// Mitsubishi GX Works2 project: 22APRIL   PLC: FX3G
// PLC project

// global labels: Global1
VAR_GLOBAL
  Work_Day_Light AT X007 : BOOL;
  Chocolate_First_Input AT D1550 : REAL;
  Chocolate_Stock AT D1350 : REAL;
  Nuts_First_Input AT D1600 : REAL;
  Nuts_Stock AT D1400 : REAL;
  Start_Day AT X007 : BOOL;
  Start AT Y007 : BOOL;
  WorkingDay AT Y007 : BOOL;
  Emergancy AT X005 : BOOL;
  Working_Day_Light AT Y007 : BOOL;
  End_Day AT M1 : BOOL;
  No_Inventory AT M2 : BOOL;
  Pistachio_First_Input AT D1700 : REAL;
  Kadaif_First_Input AT D1650 : REAL;
  Pistachio_Stock AT D1450 : REAL;
  Kadaif_Stock AT D1500 : REAL;
  Melting_Button AT X001 : BOOL;
END_VAR
VAR_GLOBAL CONSTANT
  Chocolate_Amout_Melting : REAL := 400;
END_VAR
VAR_GLOBAL
  No_Choclate AT M3 : BOOL;
  Melting_Light AT Y001 : BOOL;
  Temp_Sensor AT X002 : BOOL;
  Valid_Chocolate AT M11 : BOOL;
  No_Valid_Chocolate AT M11 : BOOL;
  Choose_Filling AT X004 : BOOL;
  Choose_Type_Analog_Input AT D8280 : INT;
END_VAR
VAR_GLOBAL CONSTANT
  const400 : REAL := 400.0;
END_VAR
VAR_GLOBAL
  Real_Undivided_Input AT D1150 : REAL;
  Real_Input AT D1250 : REAL;
  Choose_Type AT X004 : BOOL;
END_VAR
VAR_GLOBAL CONSTANT
  Constant_6 : REAL := 6;
END_VAR
VAR_GLOBAL
  Dubai_Light AT M8 : BOOL;
END_VAR
VAR_GLOBAL CONSTANT
  Constant_5 : REAL := 5;
END_VAR
VAR_GLOBAL
  Nuts_Light AT M9 : BOOL;
  Finished_Packages AT M10 : BOOL;
  Finished_Chocolate_Bar AT CC1 : BOOL;
END_VAR
VAR_GLOBAL CONSTANT
  NutsDubaiAmount : REAL := 20;
  PistachioDubaiAmount : REAL := 120;
  KadaifDubaiAmount : REAL := 60;
END_VAR
VAR_GLOBAL
  Kadai_Stock AT D1500 : REAL;
  Valid_Dubai AT M11 : BOOL;
END_VAR
VAR_GLOBAL CONSTANT
  NutsNutsAmount : REAL := 100;
  PistachioNutsAmount : REAL := 100;
END_VAR
VAR_GLOBAL
  Valid_Nuts AT M12 : BOOL;
END_VAR
VAR_GLOBAL CONSTANT
  ChocolatePackageAmount : REAL := 400;
  Chocolate_Amount_Melting : REAL := 400;
END_VAR
VAR_GLOBAL
  Melting_Container AT D1200 : REAL;
  Loction_Sensor AT X003 : BOOL;
  Constant_4 AT D8280 : INT;
END_VAR
VAR_GLOBAL CONSTANT
  const4 : INT := 40;
END_VAR
VAR_GLOBAL
  Casting_Answer AT TS2 : BOOL;
  Casting AT Y002 : BOOL;
END_VAR
VAR_GLOBAL CONSTANT
  timer4 : REAL := 4;
  const40 : INT := 40;
END_VAR
VAR_GLOBAL
  Filling_Container AT D1800 : REAL;
END_VAR
VAR_GLOBAL CONSTANT
  Dubai_Filling_Total : REAL := 200;
END_VAR
VAR_GLOBAL
  Filling AT M14 : BOOL;
  Flicker AT M6 : BOOL;
  Flicker3 AT TC4 : BOOL;
END_VAR
VAR_GLOBAL CONSTANT
  const50 : INT := 50;
END_VAR
VAR_GLOBAL
  Flicker_Timer3 AT TS4 : BOOL;
  FlickerLight3 AT Y003 : BOOL;
  Flicker4 AT TC5 : BOOL;
  Flicker_Timer4 AT TS5 : BOOL;
  FlickerLight4 AT Y004 : BOOL;
END_VAR
VAR_GLOBAL CONSTANT
  const10 : INT := 1;
END_VAR
VAR_GLOBAL
  Filling_Timer AT TS6 : BOOL;
  Flicker_Timer AT TC6 : BOOL;
  Cooling_Button AT X006 : BOOL;
  Cooling_Light AT Y006 : BOOL;
  Cooling_Final AT TS3 : BOOL;
  Cooling_Timer AT TC3 : BOOL;
END_VAR
VAR_GLOBAL CONSTANT
  const30 : INT := 30;
END_VAR
VAR_GLOBAL
  Flashing_Light AT M7 : BOOL;
  Finished_Filling_Light AT M7 : BOOL;
END_VAR
VAR_GLOBAL CONSTANT
  BarsInPackage : REAL := 4;
END_VAR
VAR_GLOBAL
  Cooling_System AT D1750 : REAL;
  Packing_One_Bar AT X000 : BOOL;
  Package_Full AT M7 : BOOL;
  OneBar_Counter AT CC0 : BOOL;
  FourBar_Count AT CC1 : BOOL;
END_VAR
VAR_GLOBAL CONSTANT
  cons4 : INT := 4;
END_VAR
VAR_GLOBAL
  Start_Count AT CS0 : BOOL;
  Stop_Count AT CS1 : BOOL;
  Packing_Light AT Y005 : BOOL;
  Finished_Packages_Container AT D1100 : REAL;
END_VAR
VAR_GLOBAL CONSTANT
  Const1 : REAL := 1;
END_VAR
VAR_GLOBAL
  New_Package_Count AT CN1 : INT;
END_VAR
VAR_GLOBAL CONSTANT
  Cons1 : REAL := 1;
END_VAR
VAR_GLOBAL
  Cooling : BOOL;
  Casting_Timer1 AT TC2 : BOOL;
  Pouring_Light1 AT M13 : BOOL;
  Casting_Time_Finish AT M14 : BOOL;
END_VAR
VAR_GLOBAL CONSTANT
  Divide_analog : REAL := 40;
END_VAR
VAR_GLOBAL
  Chocolate_package_answer AT D1470 : REAL;
  analog_output1 AT D8282 : INT;
  start_counting AT CN0 : INT;
END_VAR

// task Task_01 (event TRUE, interval 0, priority 31): POU_01

PROGRAM POU_01
VAR
  Pistachio : REAL;
  Melting : BOOL;
  Casting_Final : BOOL;
  Casting_Light : BOOL;
  Filling_Light : BOOL;
  Casting_Timer : BOOL;
  pouring_light : BOOL;
END_VAR
(* structured ladder/FBD written out as ST: instructions are called as NAME(EN, inputs, outputs); _pN, _eN, _tN stand for wires *)
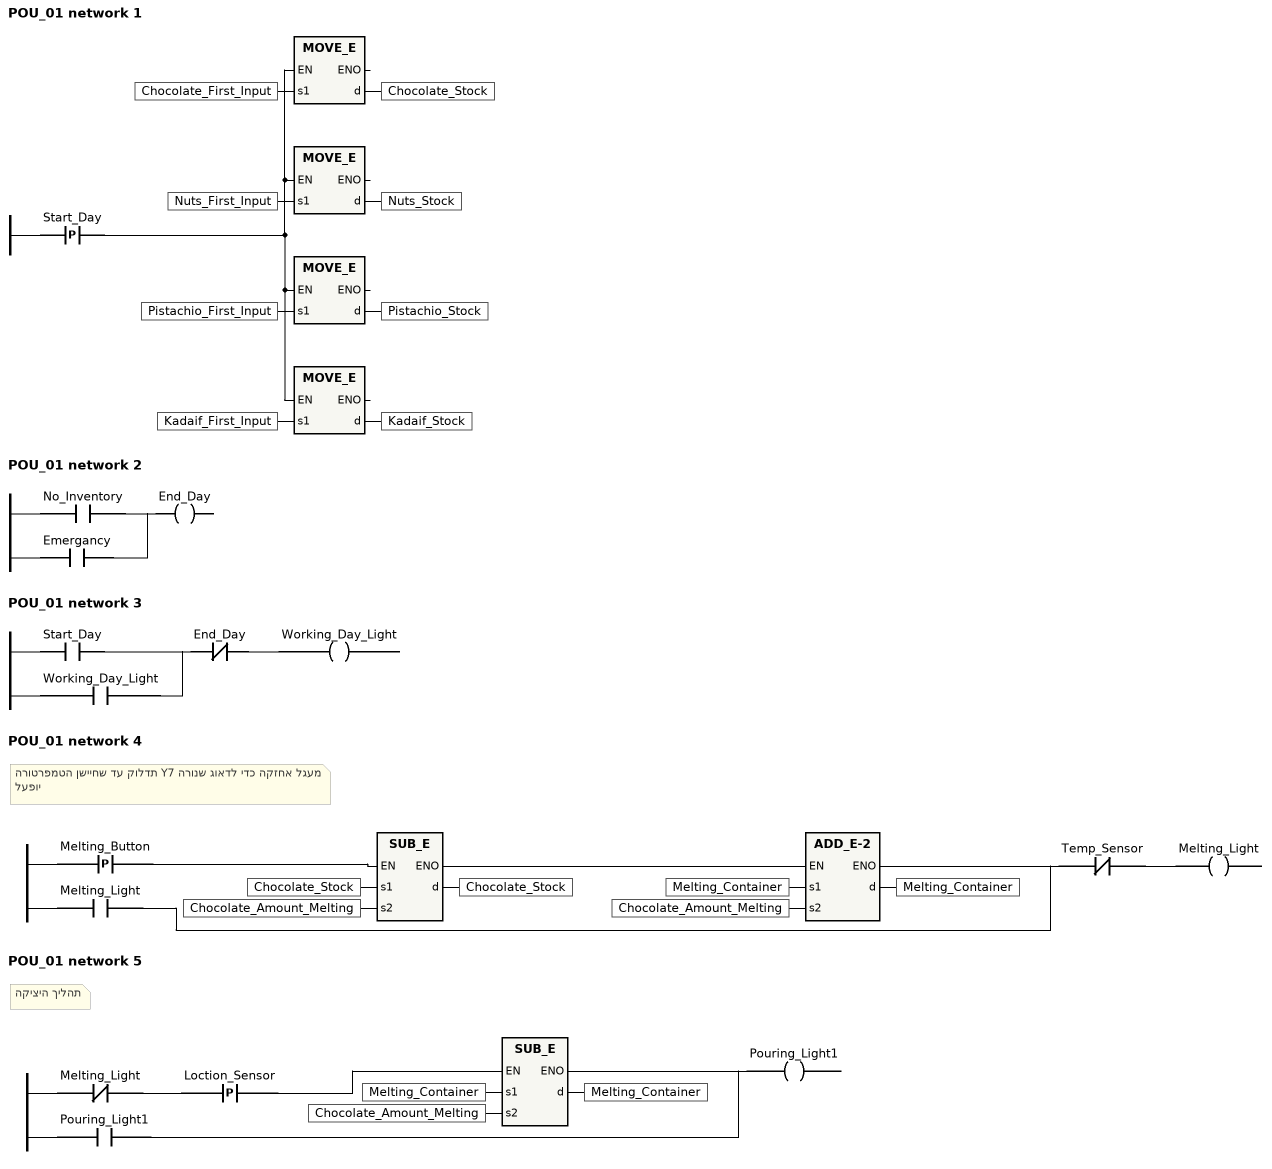
(* network 1 *)
_p1 := LDP(TRUE, Start_Day);
MOVE_E(_p1, Chocolate_First_Input, Chocolate_Stock);
MOVE_E(_p1, Nuts_First_Input, Nuts_Stock);
MOVE_E(_p1, Pistachio_First_Input, Pistachio_Stock);
MOVE_E(_p1, Kadaif_First_Input, Kadaif_Stock);
(* network 2 *)
End_Day := No_Inventory OR Emergancy;
(* network 3 *)
Working_Day_Light := (Start_Day OR Working_Day_Light) AND NOT End_Day;
(* network 4 *)
(* מעגל אחזקה כדי לדאוג שנורה Y7 תדלוק עד שחיישן הטמפרטורה יופעל *)
_e1 := SUB_E(LDP(TRUE, Melting_Button), Chocolate_Stock, Chocolate_Amount_Melting, Chocolate_Stock);
_e2 := ADD_E(_e1, Melting_Container, Chocolate_Amount_Melting, Melting_Container);
Melting_Light := (_e2 OR Melting_Light) AND NOT Temp_Sensor;
(* network 5 *)
(* תהליך היציקה *)
_e1 := SUB_E(NOT Melting_Light AND LDP(TRUE, Loction_Sensor), Melting_Container, Chocolate_Amount_Melting, Melting_Container);
Pouring_Light1 := _e1 OR Pouring_Light1;
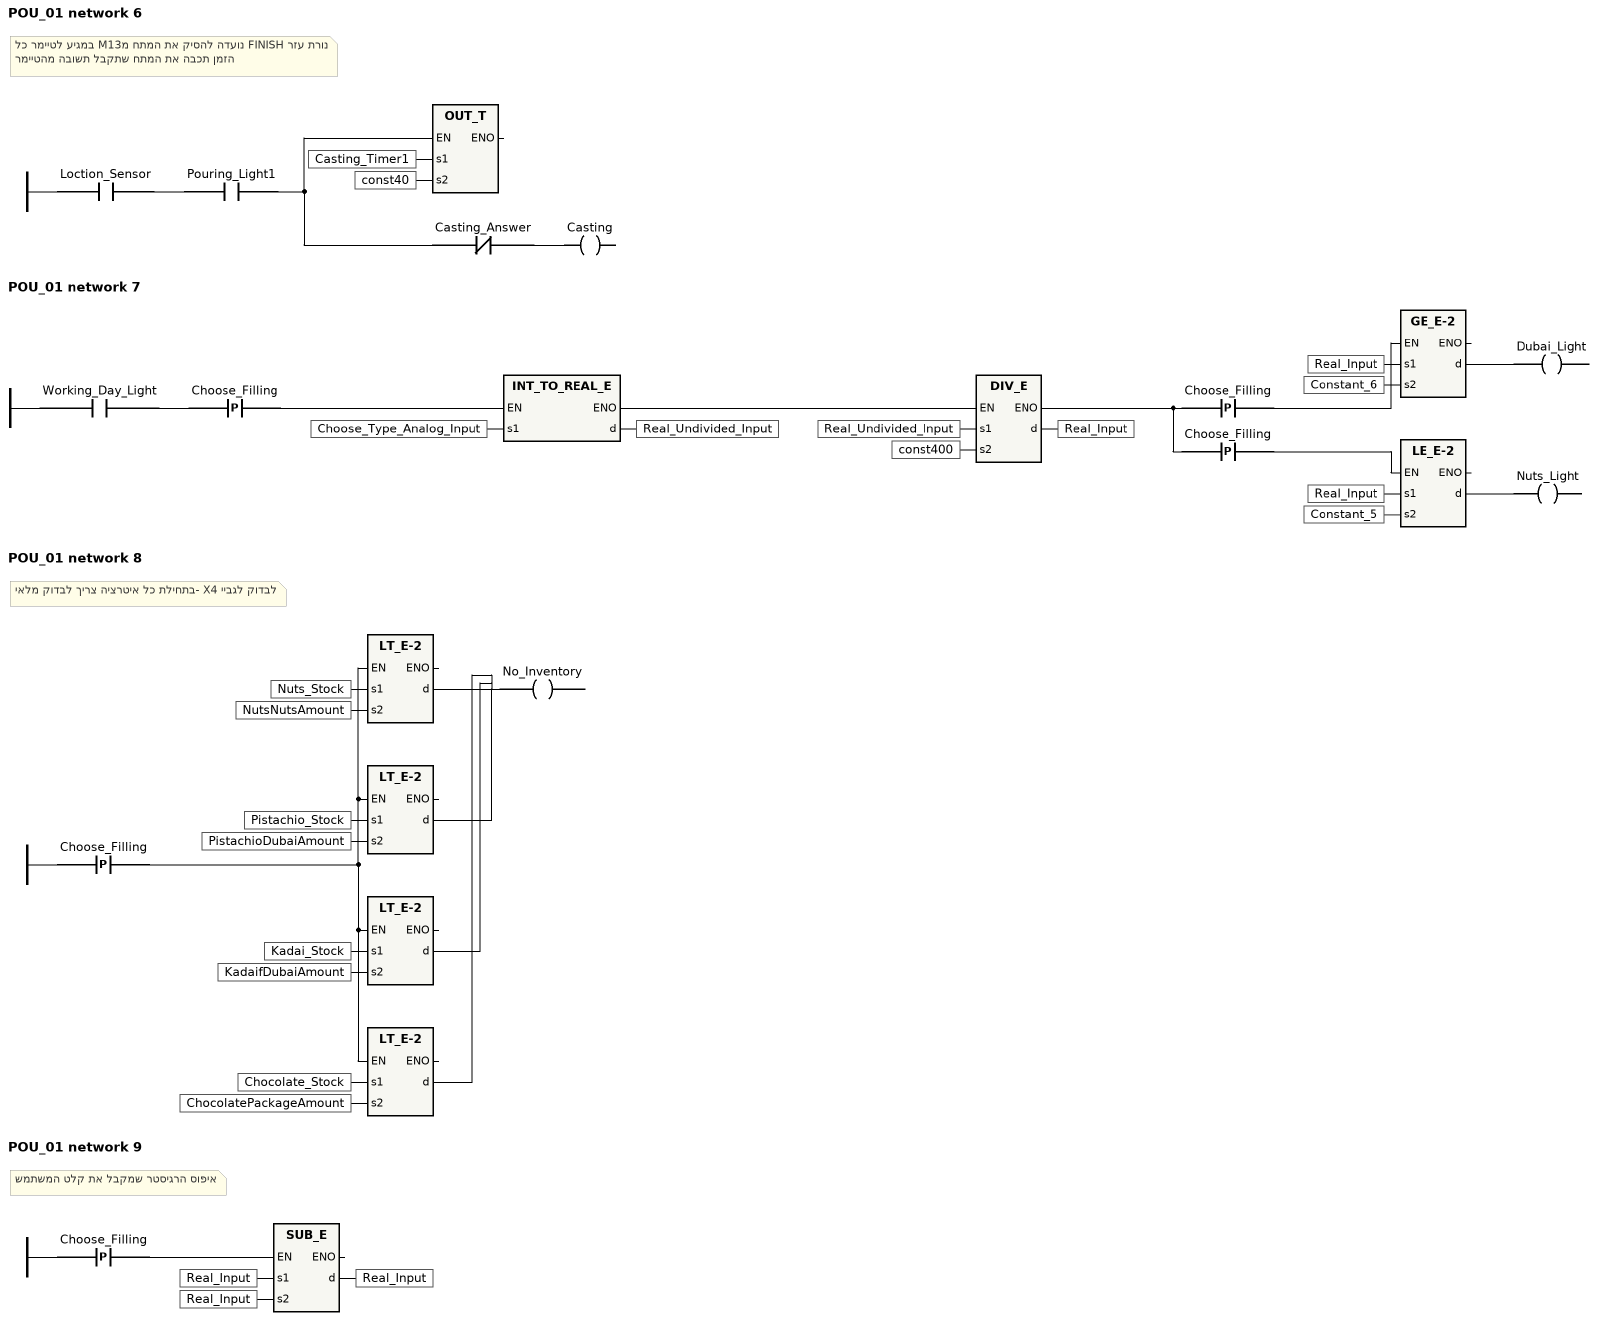
(* network 6 *)
(* נורת עזר FINISH נועדה להסיק את המתח מM13 במגיע לטיימר כל הזמן תכבה את המתח שתקבל תשובה מהטיימר *)
_p1 := Loction_Sensor AND Pouring_Light1;
OUT_T(_p1, Casting_Timer1, const40);
Casting := _p1 AND NOT Casting_Answer;
(* network 7 *)
_e1 := INT_TO_REAL_E(Working_Day_Light AND LDP(TRUE, Choose_Filling), Choose_Type_Analog_Input, Real_Undivided_Input);
_e2 := DIV_E(_e1, Real_Undivided_Input, const400, Real_Input);
GE_E(_e2 AND LDP(TRUE, Choose_Filling), Real_Input, Constant_6, _t3);
Dubai_Light := _t3;
LE_E(_e2 AND LDP(TRUE, Choose_Filling), Real_Input, Constant_5, _t4);
Nuts_Light := _t4;
(* network 8 *)
(* לבדוק לגביי X4 -בתחילת כל איטרציה צריך לבדוק מלאי *)
_p1 := LDP(TRUE, Choose_Filling);
LT_E(_p1, Nuts_Stock, NutsNutsAmount, _t2);
LT_E(_p1, Pistachio_Stock, PistachioDubaiAmount, _t3);
LT_E(_p1, Kadai_Stock, KadaifDubaiAmount, _t4);
LT_E(_p1, Chocolate_Stock, ChocolatePackageAmount, _t5);
No_Inventory := _t2 OR _t3 OR _t4 OR _t5;
(* network 9 *)
(* איפוס הרגיסטר שמקבל את קלט המשתמש *)
SUB_E(LDP(TRUE, Choose_Filling), Real_Input, Real_Input, Real_Input);
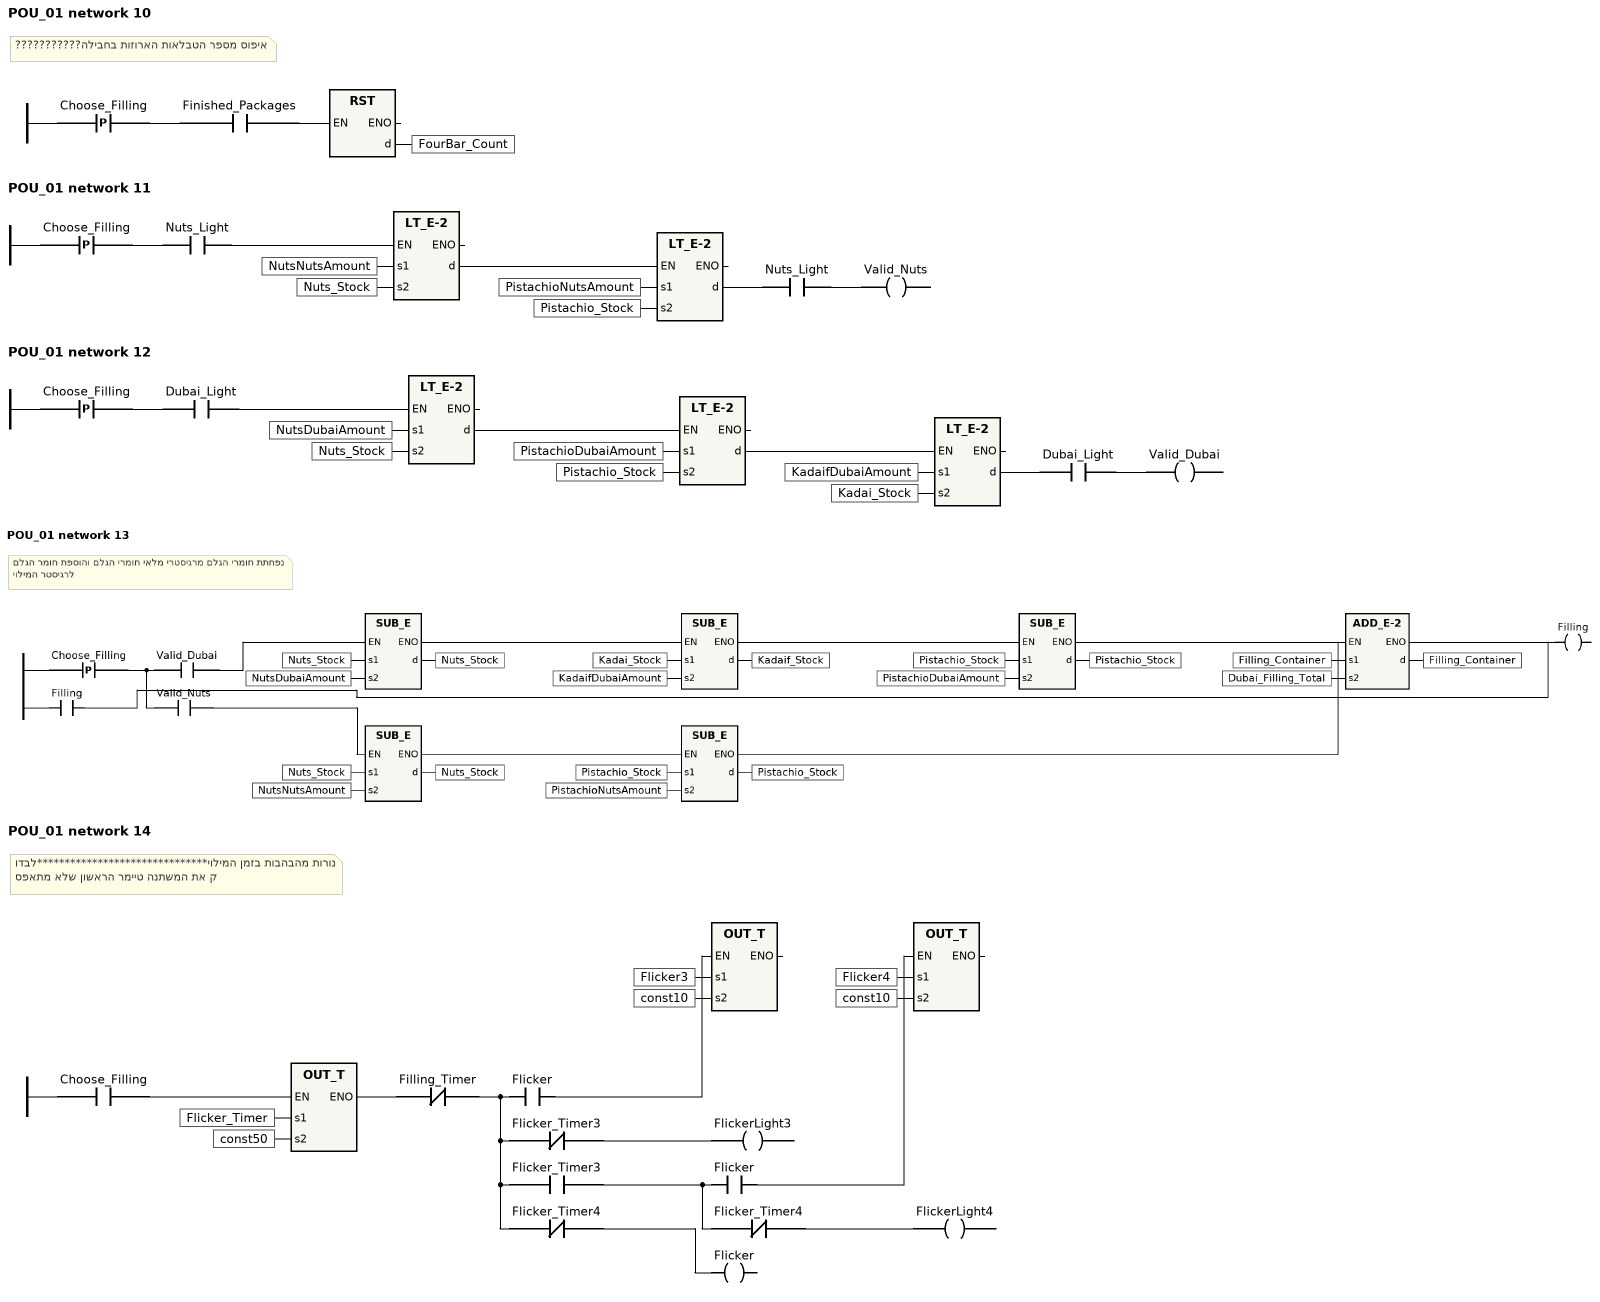
(* network 10 *)
(* איפוס מספר הטבלאות הארוזות בחבילה??????????? *)
RST(LDP(TRUE, Choose_Filling) AND Finished_Packages, FourBar_Count);
(* network 11 *)
LT_E(LDP(TRUE, Choose_Filling) AND Nuts_Light, NutsNutsAmount, Nuts_Stock, _t1);
LT_E(_t1, PistachioNutsAmount, Pistachio_Stock, _t2);
Valid_Nuts := _t2 AND Nuts_Light;
(* network 12 *)
LT_E(LDP(TRUE, Choose_Filling) AND Dubai_Light, NutsDubaiAmount, Nuts_Stock, _t1);
LT_E(_t1, PistachioDubaiAmount, Pistachio_Stock, _t2);
LT_E(_t2, KadaifDubaiAmount, Kadai_Stock, _t3);
Valid_Dubai := _t3 AND Dubai_Light;
(* network 13 *)
(* נפחתת חומרי הגלם מרגיסטרי מלאי חומרי הגלם והוספת חומר הגלם לרגיסטר המילוי *)
_p1 := LDP(TRUE, Choose_Filling);
_e2 := SUB_E(_p1 AND Valid_Dubai, Nuts_Stock, NutsDubaiAmount, Nuts_Stock);
_e3 := SUB_E(_e2, Kadai_Stock, KadaifDubaiAmount, Kadaif_Stock);
_e4 := SUB_E(_e3, Pistachio_Stock, PistachioDubaiAmount, Pistachio_Stock);
_e5 := SUB_E(_p1 AND Valid_Nuts, Nuts_Stock, NutsNutsAmount, Nuts_Stock);
_e6 := SUB_E(_e5, Pistachio_Stock, PistachioNutsAmount, Pistachio_Stock);
_e7 := ADD_E(_e4 OR _e6, Filling_Container, Dubai_Filling_Total, Filling_Container);
Filling := _e7 OR Filling;
(* network 14 *)
(* נורות מהבהבות בזמן המילוי*******************************לבדוק את המשתנה טיימר הראשון שלא מתאפס *)
_e1 := OUT_T(Choose_Filling, Flicker_Timer, const50);
_p2 := _e1 AND NOT Filling_Timer;
OUT_T(_p2 AND Flicker, Flicker3, const10);
FlickerLight3 := _p2 AND NOT Flicker_Timer3;
_p3 := _p2 AND Flicker_Timer3;
OUT_T(_p3 AND Flicker, Flicker4, const10);
FlickerLight4 := _p3 AND NOT Flicker_Timer4;
Flicker := _p2 AND NOT Flicker_Timer4;
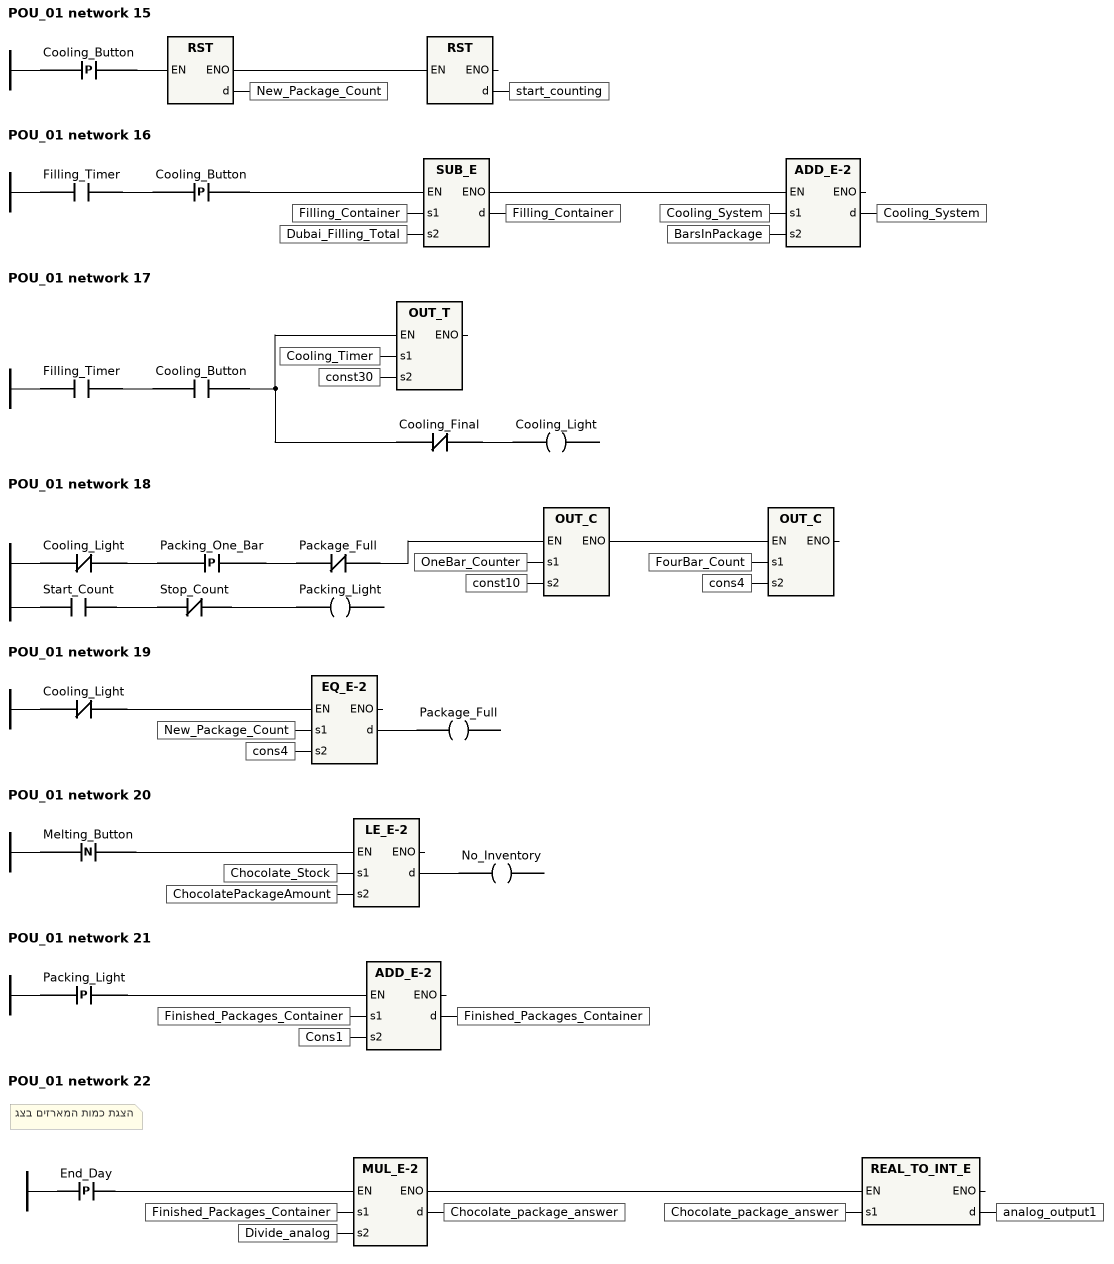
(* network 15 *)
_e1 := RST(LDP(TRUE, Cooling_Button), New_Package_Count);
RST(_e1, start_counting);
(* network 16 *)
_e1 := SUB_E(Filling_Timer AND LDP(TRUE, Cooling_Button), Filling_Container, Dubai_Filling_Total, Filling_Container);
ADD_E(_e1, Cooling_System, BarsInPackage, Cooling_System);
(* network 17 *)
_p1 := Filling_Timer AND Cooling_Button;
OUT_T(_p1, Cooling_Timer, const30);
Cooling_Light := _p1 AND NOT Cooling_Final;
(* network 18 *)
_e1 := OUT_C(NOT Cooling_Light AND LDP(TRUE, Packing_One_Bar) AND NOT Package_Full, OneBar_Counter, const10);
OUT_C(_e1, FourBar_Count, cons4);
Packing_Light := Start_Count AND NOT Stop_Count;
(* network 19 *)
EQ_E(NOT Cooling_Light, New_Package_Count, cons4, _t1);
Package_Full := _t1;
(* network 20 *)
LE_E(LDF(TRUE, Melting_Button), Chocolate_Stock, ChocolatePackageAmount, _t1);
No_Inventory := _t1;
(* network 21 *)
ADD_E(LDP(TRUE, Packing_Light), Finished_Packages_Container, Cons1, Finished_Packages_Container);
(* network 22 *)
(* הצגת כמות המארזים בצג *)
_e1 := MUL_E(LDP(TRUE, End_Day), Finished_Packages_Container, Divide_analog, Chocolate_package_answer);
REAL_TO_INT_E(_e1, Chocolate_package_answer, analog_output1);
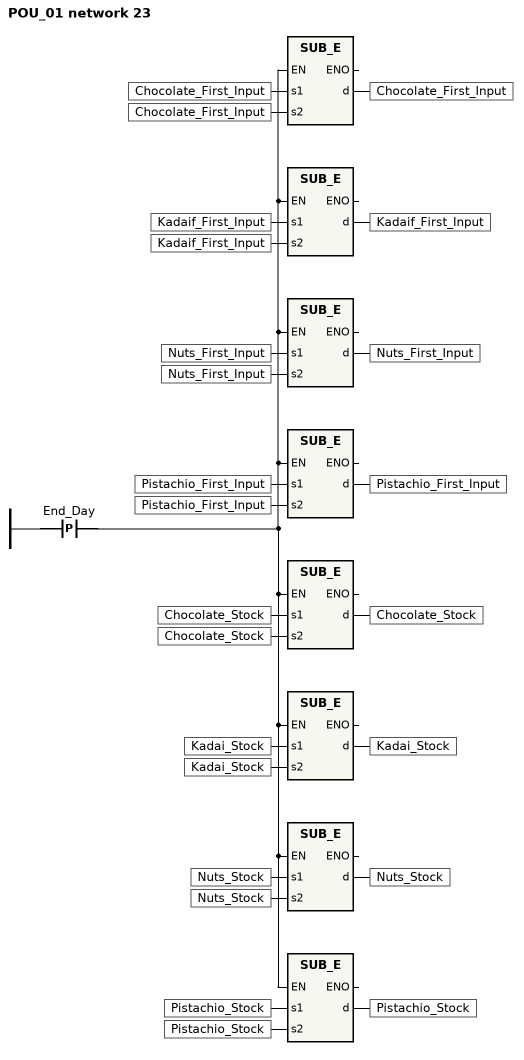
(* network 23 *)
_p1 := LDP(TRUE, End_Day);
SUB_E(_p1, Chocolate_First_Input, Chocolate_First_Input, Chocolate_First_Input);
SUB_E(_p1, Kadaif_First_Input, Kadaif_First_Input, Kadaif_First_Input);
SUB_E(_p1, Nuts_First_Input, Nuts_First_Input, Nuts_First_Input);
SUB_E(_p1, Pistachio_First_Input, Pistachio_First_Input, Pistachio_First_Input);
SUB_E(_p1, Chocolate_Stock, Chocolate_Stock, Chocolate_Stock);
SUB_E(_p1, Kadai_Stock, Kadai_Stock, Kadai_Stock);
SUB_E(_p1, Nuts_Stock, Nuts_Stock, Nuts_Stock);
SUB_E(_p1, Pistachio_Stock, Pistachio_Stock, Pistachio_Stock);
END_PROGRAM
